{attribute 'pack_mode' := '1'}
TYPE ChangeAxisEnable EXTENDS IncomingMessage :
STRUCT
	axisIndex: INT; (* 1 or 2.*)
	enabled: BOOL;
END_STRUCT
END_TYPE

(* stored: Version 1.1.0.1, ProductVersion 3.1.4022.12
   DUT ChangeAxisEnable: Id {e2ff3d12-a148-4208-bc86-130983783fa1} *)
